// Gets the upper bound index of the array of specified type.
FUNCTION F_GetByteArrayUpperBound : T_Position // The upper bound index of the specified array.
VAR_IN_OUT
	arArray : ARRAY[*] OF BYTE; // The array to query.
END_VAR

F_GetByteArrayUpperBound := UPPER_BOUND(arArray, 1);

END_FUNCTION

(* stored: Version 1.1.0.1
   POU F_GetByteArrayUpperBound: Id {9d42bde0-de67-0e77-07f3-78c0e93ee27a}, SpecialFunc None *)
